FUNCTION_BLOCK FB_WORD_TO_BYTES IMPLEMENTS I_WORD_TO_BYTES
VAR_INPUT
END_VAR
VAR_OUTPUT
END_VAR
VAR
	uWordToBytes:				U_BytesToWord ;
//Für Input
	bBytesOut1					AT %Q* :BYTE;
	bBytesOut2					AT %Q* :BYTE;
	lrWordIn:					LREAL;	
	
	lrUnscaledIn:				LREAL;
	lrScaledIn:					LREAL;
	temp_gain:					LREAL;
	temp_offset:				LREAL;
	lrX_Max:					LREAL	:=1;
	lrX_Min:					LREAL;
	lrY_Max:					LREAL	:=1;
	lrY_Min:					LREAL;	
	i:							INT;
END_VAR

METHOD FB_init : BOOL
VAR_INPUT
	bInitRetains : 				BOOL; // if TRUE, the retain variables are initialized (warm start / cold start)
	bInCopyCode : 				BOOL;  // if TRUE, the instance afterwards gets moved into the copy code (online change)
END_VAR
END_METHOD

(*=== Method: M_Run  ============================================

 @brief: Here is the global code (Timer, Event, Flange,...)*)
METHOD M_Run

VAR
END_VAR
i:=i+1;

uWordToBytes.uintOut:=LREAL_TO_WORD(lrWordIn);
bBytesOut2:=uWordToBytes.arByteIn[0];
bBytesOut1:=uWordToBytes.arByteIn[1];

IF lrY_Max = 0 THEN
	lrY_Max:=1;
END_IF
IF lrX_Max =0 THEN
	lrX_Max:=1;
END_IF

// Ausgang Scallieren
temp_gain := (lrY_Max - lrY_Min) / (lrX_Max - lrX_Min);
temp_offset := lrY_Min - lrX_Min * temp_gain;
lrWordIn := lrUnscaledIn * temp_gain + temp_offset;

IF lrUnscaledIn > lrX_Max THEN
    lrWordIn := REAL_TO_INT(lrY_Max);
ELSIF lrUnscaledIn < lrX_Min THEN
    lrWordIn := REAL_TO_INT(lrY_Min);
END_IF;
END_METHOD

(*=== Property: P_Event  ============================================

 @param [set]: 	Set the Structure "ST_EVENT" from another Object
 @param [get]: 	Return the Structure "ST_EVENT", it contains the actual 
					event of the Object *)
PROPERTY P_Event : GenLib.ST_EVENT
GET
END_GET
SET
END_SET
END_PROPERTY

(*=== Property: P_FullObjectPath  ============================================

 @param [set]: 	Set the Object Path (Clear String of Object)
 @param [get]: 	Return the Objectpath *)
PROPERTY P_FullObjectPath : STRING
GET
END_GET
SET
END_SET
END_PROPERTY

(*=== Property: P_Global_Ack  ============================================

 @param [set]: 	Set the Bit for Ack from another Object
 @param [get]: 	Return the state of Ack Bit*)
PROPERTY P_Global_Ack : BOOL
GET
END_GET
SET
END_SET
END_PROPERTY

(*=== Property: P_GlobalID  ============================================

 @param [set]: 	-
 @param [get]: 	Return the string of instance path*)
PROPERTY P_GlobalID : STRING
GET
END_GET
END_PROPERTY

PROPERTY P_VALUE : LREAL
GET
P_VALUE:=lrUnscaledIn;
END_GET
SET
lrUnscaledIn:=P_VALUE;
END_SET
END_PROPERTY

PROPERTY P_X_MAX : LREAL
GET
P_X_MAX:=lrX_Max;
END_GET
SET
lrX_Max:=P_X_MAX;
END_SET
END_PROPERTY

PROPERTY P_X_MIN : LREAL
GET
P_X_MIN:=lrX_Min;
END_GET
SET
lrX_Min:=P_X_MIN;
END_SET
END_PROPERTY

PROPERTY P_Y_MAX : LREAL
GET
P_Y_MAX:=lrY_Max;
END_GET
SET
lrY_Max:=P_Y_MAX;
END_SET
END_PROPERTY

PROPERTY P_Y_MIN : LREAL
GET
P_Y_MIN:=lrY_Min;
END_GET
SET
lrY_Min:=P_Y_MIN;
END_SET
END_PROPERTY

END_FUNCTION_BLOCK

(* stored: Version 1.1.0.1, ProductVersion 3.1.4024.9
   POU FB_WORD_TO_BYTES: Id {6fb4d424-b85e-4656-9157-5c9d3697dbac}, SpecialFunc None
   Method FB_init: Id {6e4fef96-38dc-4d12-b309-39071f70273c}
   Method M_Run: Id {be110074-6538-4c16-8154-8fbd357f8f5a}
   Property P_Event: Id {959872e2-20d3-415a-8d51-094ea9d87d14}
   Get Get: Id {1c52330a-4e00-4ed9-8165-c783c7a42453}
   Set Set: Id {d8c6f6ad-d9a1-44c4-989c-5178b7481474}
   Property P_FullObjectPath: Id {50020da1-24cb-458e-a809-1d59001dab7f}
   Get Get: Id {a69ef8e5-3486-4247-aa57-c9370be7d699}
   Set Set: Id {bc4ef5d5-821f-448a-9b96-67b0901d975b}
   Property P_Global_Ack: Id {a01ef1b9-1066-46bb-b48e-01067b863964}
   Get Get: Id {ba7a612a-1978-4f61-92a4-46b9f550a528}
   Set Set: Id {e8d821d6-a558-4994-937f-7d921034c2e5}
   Property P_GlobalID: Id {0d4d9fb4-25bd-4d5b-849e-a2c682484e3d}
   Get Get: Id {dd8482fd-3005-401f-b045-b5e3e91d50c5}
   Property P_VALUE: Id {b5800c6d-741d-44a2-b8f5-1a9e597f0e0d}
   Get Get: Id {1cd53712-ad47-413d-ad19-d3c3e15265a6}
   Set Set: Id {93e3b863-ae6b-4d75-bf0a-0c2441f0a531}
   Property P_X_MAX: Id {4f57cb83-22c2-4303-a2ff-383e0e6fe3d2}
   Get Get: Id {49cb7143-8cd3-4379-8db2-37a5511fdf17}
   Set Set: Id {0b8044bd-ec70-4732-8428-8d5fe4e191bc}
   Property P_X_MIN: Id {4d01d0e0-1f3c-4c18-8727-5630bd256924}
   Get Get: Id {17dceb25-8964-40d3-ae76-bea13d0c9888}
   Set Set: Id {4e26a83d-efaa-4612-a74b-4dfba0c486ea}
   Property P_Y_MAX: Id {13609b42-00be-45a4-83f2-21a01cda2bef}
   Get Get: Id {af0c1340-2e2d-440a-933c-ba03d70adc78}
   Set Set: Id {9eb9331b-b39c-4acf-8d28-7ed29ec260d7}
   Property P_Y_MIN: Id {01234699-7865-4fb1-8c63-45a83674e0a9}
   Get Get: Id {c2e9b16e-6ff6-40c1-b3a3-10e914db1239}
   Set Set: Id {c56ad86c-2a3d-4cee-92af-9ea339f77116} *)
